{attribute addProperty BoxType "ATH2000-0250-0023"}
{attribute addProperty Id "A_0015_ATH2040_5250_0022ATH2040_948A301E9812.25"}
{attribute addProperty CRC "3607143149"}
{attribute addProperty SizeInBites "98"}
{attribute addProperty SizeInBytes "12.25"}
TYPE A_0002_ATH2000_0250_0023_D700A2ED EXTENDS ATH2000_BA5A9548 :
STRUCT
	{attribute addProperty Name "A_0015_ATH2040_5250_0022"}
	A_0015_ATH2040_5250_0022 : ATH2040_948A301E;
END_STRUCT
END_TYPE

(* stored: Version 1.2.0.0, ProductVersion 3.1.4024.9
   DUT A_0002_ATH2000_0250_0023_D700A2ED: Id {77233b33-1079-4382-b48a-32b6d7a1bf26} *)
